ABB RobotStudio station: Palletizing_Rapids_programming.rspag

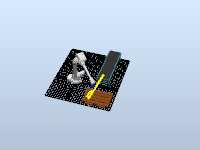
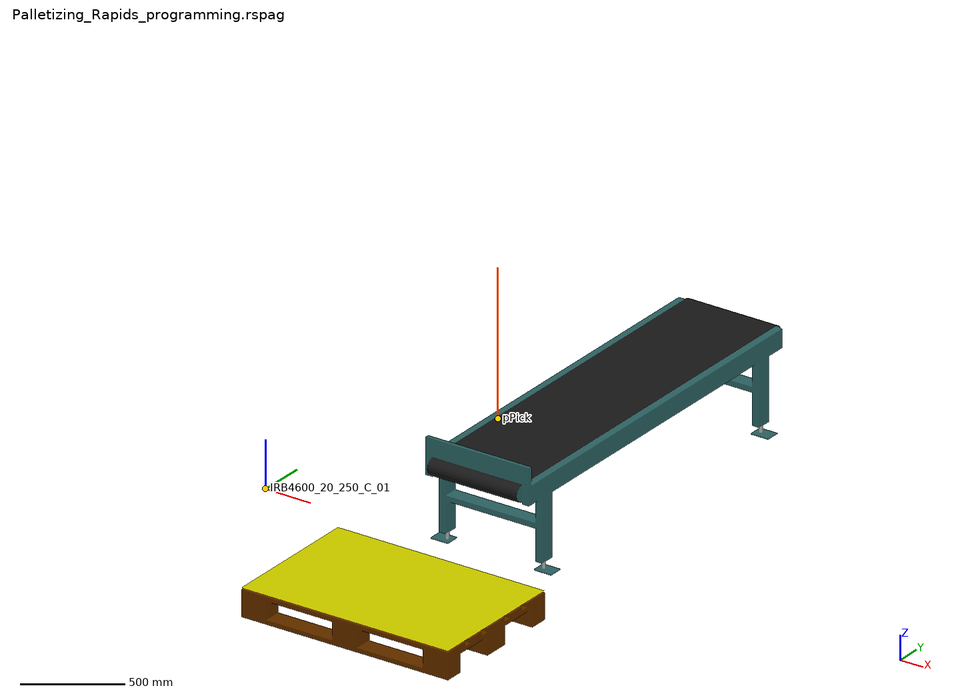
[picture v1: parts stored in the station drawn from their meshes, with robot base, taught points and paths (robot models come from the ABB library and are not in the file)]
--- station ---
Station palletizing (saved by RobotStudio 21.2.9526.0)
Controller IRB4600
  mechanical unit ROB_1: IRB4600_20_250_C_01, 6 joints, base frame (0, 0, 0) mm
Layout (positions relative to the parent item):
  - IRB4600_20_250_C_01 [mechanism, from Robots\IRB4600_20_250_C_G_01.rslib] at (0, 0, 0) mm; joint values [-0.6905, 0.1476, 0.3704, 0, 1.0528, -0.6905] (rad or m)
  - Belt Conveyor [part], size 703.5 x 2188.6 x 501 mm
  - Box [part], size 500 x 300 x 200 mm
  - SC_InFeeder [smart component]
      signals: DO doBoxInPos
      connections:
        LineSensor.SensorOut -> SC_InFeeder.doBoxInPos
        LineSensor.SensorOut -> LogicGate_2.InputA
        LogicGate_2.Output -> Source.Execute
    - Source [smart component, from Components\Source.rslib]
        properties: Source=Box; Copy=(none); Parent=(none); Position=[0 0 0]; Orientation=[0 0 0]; Transient=true; PhysicsBehavior=3
    - LineSensor [smart component, from Components\LineSensor.rslib]
        properties: Start=[1.3 -0.09 0.547]; End=[1.3 -0.03 0.547]; Radius=0; SensedPart=(none); SensedPoint=[0 0 0]
      - _sensorPart_ [part], size 0 x 60 x 0 mm
    - LogicGate_2 [smart component, from Components\LogicGate.rslib]
        properties: Operator=NOT; Delay=0
  - Belt [part], size 529.1 x 2200.3 x 102.1 mm
  - Stop [part], size 600 x 20 x 100 mm
  - SC_VacuumTool [smart component] at (1150, -950.15, 1035.93) mm, rotated rx 180 ry 0 rz 180 deg
      signals: DI diAttach, DO doAttached
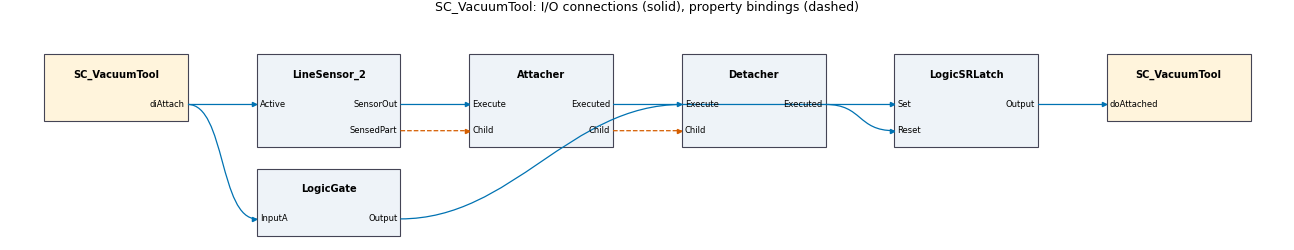
      connections:
        SC_VacuumTool.diAttach -> LineSensor_2.Active
        LineSensor_2.SensorOut -> Attacher.Execute
        Attacher.Executed -> LogicSRLatch.Set
        SC_VacuumTool.diAttach -> LogicGate.InputA
        LogicGate.Output -> Detacher.Execute
        Detacher.Executed -> LogicSRLatch.Reset
        LogicSRLatch.Output -> SC_VacuumTool.doAttached
        LineSensor_2.SensedPart => Attacher.Child
        Attacher.Child => Detacher.Child
    - LineSensor_2 [smart component, from Components\LineSensor.rslib]
        properties: Start=[0 0 0.1122]; End=[0 0 0.16]; Radius=0; SensedPart=(none); SensedPoint=[1.20967431640625 -0.544369445800781 1.13760888671875]
      - _sensorPart_ [part], size 0 x 0 x 47.8 mm
    - Attacher [smart component, from Components\Attacher.rslib]
        properties: Parent=Vacuum Tool; Flange=0; Child=(none); Mount=false; Offset=[0 0 0]; Orientation=[0 0 0]
    - Detacher [smart component, from Components\Detacher.rslib]
        properties: Child=(none); KeepPosition=true
    - LogicGate [smart component, from Components\LogicGate.rslib]
        properties: Operator=NOT; Delay=0
    - LogicSRLatch [smart component, from Components\LogicSRLatch.rslib]
    - Vacuum Tool [mechanism] at (0, 0, 0) mm
        TCP tVacuum at (0, 0, 150) mm
        links: Vacuum Tool
  - SC_OutFeeder [smart component]
      connections:
        PlaneSensor.SensorOut -> LogicGate.InputA
        LogicGate.Output -> Sink.Execute
    - EPAL Euro pallet [part] at (1900, -1199.98, 0) mm, rotated rx 0 ry 0 rz 90.01 deg, size 804.4 x 1206.6 x 151.6 mm
    - PlaneSensor [smart component, from Components\PlaneSensor.rslib]
        properties: Origin=[0.7 -1.2 0.154]; Axis1=[1.2 0 0]; Axis2=[0 0.8 0]; SensedPart=(none)
      - _sensorPart_ [part], size 1200 x 800 x 0 mm
    - Sink [smart component, from Components\Sink.rslib]
        properties: Object=(none)
    - LogicGate [smart component, from Components\LogicGate.rslib]
        properties: Operator=NOP; Delay=2
Attachment: SC_VacuumTool is attached to IRB4600_20_250_C_01 / Link6
Station logic (signal -> signal, property => property):
  SC_VacuumTool.doAttached -> IRB4600.diVacuum
  IRB4600.doVacuum -> SC_VacuumTool.diAttach
  SC_InFeeder.doBoxInPos -> IRB4600.diBoxInPos
Targets, tools, work objects and paths stored in the station and not in the controller backup, written as RAPID:
! task T_ROB1
MODULE Module1
  PROC PickPart()
    MoveL pPick,v300,fine,tVacuum\WObj:=wobjInFeeder;
    MoveL BOX_1,v300,fine,tVacuum\WObj:=wobjInFeeder;
    MoveL BOX_2,v300,fine,tVacuum\WObj:=wobjInFeeder;
    MoveL BOX_3,v300,fine,tVacuum\WObj:=wobjInFeeder;
    MoveL Box_4,v300,fine,tVacuum\WObj:=wobjInFeeder;
  ENDPROC
ENDMODULE


--- Backups/IRB4600/RAPID/TASK1/PROGMOD/CalibData.mod ---
MODULE CalibData
	PERS tooldata tVacuum:=[TRUE,[[0,0,150],[1,0,0,0]],[9,[0,0,100],[1,0,0,0],0,0,0]];
	TASK PERS wobjdata wobjInFeeder:=[FALSE,TRUE,"",[[0,0,0],[1,0,0,0]],[[1000,-80,497],[1,0,0,0]]];
ENDMODULE

--- Backups/IRB4600/RAPID/TASK1/PROGMOD/Module1.mod ---
MODULE Module1
    CONST robtarget pPick:=[[300.023,150,209.481],[0,-0.707106781,0.707106781,0],[0,0,0,0],[9E+09,9E+09,9E+09,9E+09,9E+09,9E+09]];
    CONST robtarget BOX_1:=[[-50,-970,-353],[0,-0.707106781,0.707106781,0],[-1,0,-2,0],[9E+09,9E+09,9E+09,9E+09,9E+09,9E+09]];
    CONST robtarget BOX_2:=[[-150.116,-570.154,-353],[0,0,1,0],[-1,0,-1,0],[9E+09,9E+09,9E+09,9E+09,9E+09,9E+09]];
    CONST robtarget BOX_3:=[[-50.116,-470.154,-353],[0,-0.707106781,0.707106781,0],[-1,0,-2,0],[9E+09,9E+09,9E+09,9E+09,9E+09,9E+09]];
    CONST robtarget Box_4:=[[-150,-870.154,-353],[0,0,1,0],[-1,0,-2,0],[9E+09,9E+09,9E+09,9E+09,9E+09,9E+09]];







    PROC main()
            Arrange_Box(5); !Enter the number of layers of boxes you want to stack.
    ENDPROC

    PROC Arrange_Box(num Levels)  !Procedure to arrange the box layers
        VAR num Odd_Eve:=1;       !holds the value to tell if layer is odd or even.
        FOR i FROM 1 TO Levels DO       !loop to stack boxes in all levels
            IF (Odd_Eve MOD 2) = 1 THEN  !If ODD layer, then stack boxes like this....

                !ODD PALLET Layer                (Total 6 boxes in each layer, 2 vertical and 4 horizontal)
                Vert_BOX 0,200*Odd_Eve,BOX_1;    !Procedure to arrange boxes in vertical order
                                                 !It takes offset, height offset(given by height of box*layer number), Target location.
                Vert_BOX 700,200*Odd_Eve,BOX_1;

                HOR_BOX 0,200*Odd_Eve,BOX_2;     !Procedure to arrange boxes in vertical order, Follows same idea as in Vert_BOX procedure.
                HOR_BOX 300,200*Odd_Eve,BOX_2;
                HOR_BOX 600,200*Odd_Eve,BOX_2;
                HOR_BOX 900,200*Odd_Eve,BOX_2;
            ELSE                                 !Else it is Even layer, then stack boxes like this....
                !EVEN PALLET Layer               (Total 6 boxes in each layer, 4 horizontal, 2 vertical)
                HOR_BOX 0,200*Odd_Eve,BOX_4;
                HOR_BOX 300,200*Odd_Eve,BOX_4;
                HOR_BOX 600,200*Odd_Eve,BOX_4;
                HOR_BOX 900,200*Odd_Eve,BOX_4;
                Vert_BOX 0,200*Odd_Eve,BOX_3;
                Vert_BOX 700,200*Odd_Eve,BOX_3;

            ENDIF
            Odd_Eve:=Odd_Eve+1;                 !Increase the level counter.
        ENDFOR
    ENDPROC


    PROC Vert_BOX(num spacing,num Z_offset, robtarget TGT)  !takes spacing offset between each box, height at which box is stacked, target location.
        VAR robtarget TOP;                                  !Dynamic variable
        VAR robtarget B1;

        TOP:=Offs(TGT,0+spacing,0,350+Z_offset);            !stores coordinates to move gripper extra 350mm from z height so that gripper comes from top.
        B1:=Offs(TGT,0+spacing,0,0+Z_offset);               !stores coordinates to move gripper to exact location.

        MoveJ Offs(pPick,0,0,800),v1000,z1,tVacuum\WObj:=wobjInFeeder;  !** The robot moves to a wait position 800 mm above the pick position. **
        WaitDI diBoxInPos,1; !** The robot waits for a box to pick at the infeeder stop. **
        MoveL pPick,v1000,fine,tVacuum\WObj:=wobjInFeeder; !** The robot goes to the pick position. **
        SetDO doVacuum,1; !** To attach the box, the robot turns on the digital output signal "doVacuum" which is connected to the Smart Component "SC_VacuumTool". **

        MoveL Offs(pPick,0,0,800),v1000,z1,tVacuum\WObj:=wobjInFeeder;
        MoveL TOP,v1000,z0,tVacuum\WObj:=wobjInFeeder;
        MoveL B1,v1000,z0,tVacuum\WObj:=wobjInFeeder;
        WaitTime 1;
        SetDO doVacuum,0;
        WaitTime 0.5;

    ENDPROC

    PROC HOR_BOX(num spacing, num Z_offset, robtarget TGT)
        VAR robtarget TOP;
        VAR robtarget B1;

        TOP:=Offs(TGT,0+spacing,0,350+Z_offset);
        B1:=Offs(TGT,0+spacing,0,0+Z_offset);

        MoveJ Offs(pPick,0,0,800),v1000,z1,tVacuum\WObj:=wobjInFeeder;
        WaitDI diBoxInPos,1;
        MoveL pPick,v1000,fine,tVacuum\WObj:=wobjInFeeder;
        SetDO doVacuum,1;

        MoveL Offs(pPick,0,0,800),v1000,z1,tVacuum\WObj:=wobjInFeeder;
        MoveL TOP,v1000,z0,tVacuum\WObj:=wobjInFeeder;
        MoveL B1,v1000,z0,tVacuum\WObj:=wobjInFeeder;
        WaitTime 1;
        SetDO doVacuum,0;
        WaitTime 0.5;
    ENDPROC
ENDMODULE

--- Backups/IRB4600/SYSPAR/EIO.cfg ---
EIO:CFG_1.0:6:1::
#
EIO_SIGNAL:

      -Name "doVacuum" -SignalType "DO" -Access "All"

      -Name "diVacuum" -SignalType "DI" -Access "All"

      -Name "diBoxInPos" -SignalType "DI" -Access "All"
